FUNCTION_BLOCK IEEE1451_SENSOR_CONTINUOUS
  {SET_ATTRIBUTE(OpcUa, DEVICE.SENSOR)}
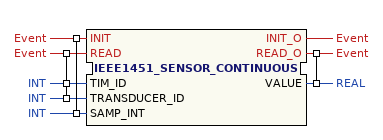
  EVENT_INPUT
    INIT WITH SAMP_INT; (* FB Initialization *)
    READ WITH TIM_ID, TRANSDUCER_ID; (* Read Sensor Request *)
  END_EVENT
  EVENT_OUTPUT
    INIT_O; (* Initialization Confirm *)
    READ_O WITH VALUE; (* Read Request Confirm *)
  END_EVENT
  VAR_INPUT
    TIM_ID : INT; (* TIM Identification *)
    TRANSDUCER_ID : INT; (* Transducer Identification *)
    SAMP_INT : INT; (* Sampling Interval *)
  END_VAR
  VAR_OUTPUT
    VALUE : REAL; (* Read Result *)
  END_VAR
END_FUNCTION_BLOCK
